% RSLogix 500 project I2P JOB 12-CAYLEN  JOHNSON.RSS, saved by version 10.00.00.00 %
PROJECT "ML06B"    % processor: Bul.1763 MicroLogix 1100 Series B %

PROGRAM FILES
  LAD 2   8 rungs

DATA FILES
  O0 OUTPUT  4 elements
  I1 INPUT  6 elements
  S2 STATUS  66 elements
  B3 BINARY  1 elements
  T4 TIMER  1 elements
  C5 COUNTER  1 elements
  R6 CONTROL  1 elements
  N7 INTEGER  1 elements
  F8 FLOAT  1 elements

LADDER 2
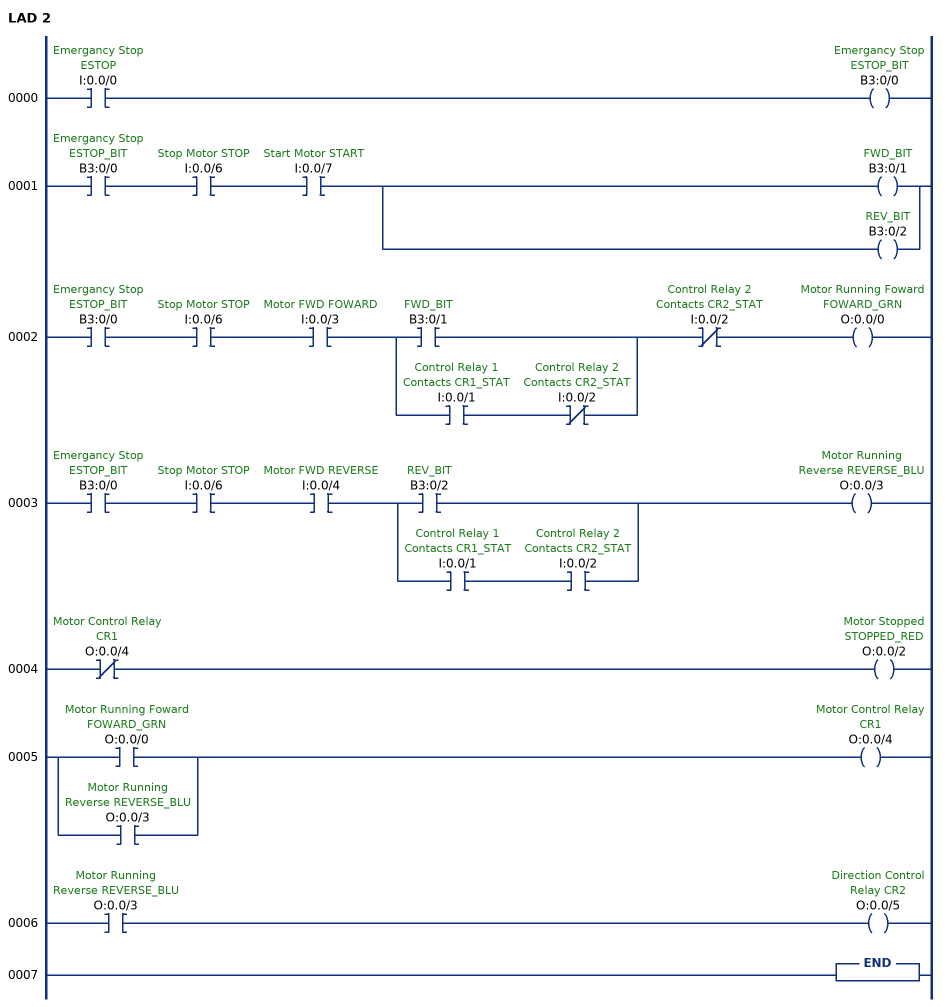
% Rung: 0 %
SOR XIC I:0.0/0 OTE B3:0/0 EOR
%   I:0.0/0  ESTOP  "Emergancy Stop" %
%   B3:0/0  ESTOP_BIT  "Emergancy Stop" %
% Rung: 1 %
SOR XIC B3:0/0 XIC I:0.0/6 XIC I:0.0/7 BST OTE B3:0/1 NXB OTE B3:0/2 BND EOR
%   B3:0/0  ESTOP_BIT  "Emergancy Stop" %
%   I:0.0/6  STOP  "Stop Motor" %
%   I:0.0/7  START  "Start Motor" %
%   B3:0/1  FWD_BIT %
%   B3:0/2  REV_BIT %
% Rung: 2 %
SOR XIC B3:0/0 XIC I:0.0/6 XIC I:0.0/3 BST XIC B3:0/1 NXB XIC I:0.0/1 XIO I:0.0/2 BND XIO I:0.0/2 OTE O:0.0/0 EOR
%   B3:0/0  ESTOP_BIT  "Emergancy Stop" %
%   I:0.0/6  STOP  "Stop Motor" %
%   I:0.0/3  FOWARD  "Motor FWD" %
%   B3:0/1  FWD_BIT %
%   I:0.0/1  CR1_STAT  "Control Relay 1 Contacts" %
%   I:0.0/2  CR2_STAT  "Control Relay 2 Contacts" %
%   O:0.0/0  FOWARD_GRN  "Motor Running Foward" %
% Rung: 3 %
SOR XIC B3:0/0 XIC I:0.0/6 XIC I:0.0/4 BST XIC B3:0/2 NXB XIC I:0.0/1 XIC I:0.0/2 BND OTE O:0.0/3 EOR
%   B3:0/0  ESTOP_BIT  "Emergancy Stop" %
%   I:0.0/6  STOP  "Stop Motor" %
%   I:0.0/4  REVERSE  "Motor FWD" %
%   B3:0/2  REV_BIT %
%   I:0.0/1  CR1_STAT  "Control Relay 1 Contacts" %
%   I:0.0/2  CR2_STAT  "Control Relay 2 Contacts" %
%   O:0.0/3  REVERSE_BLU  "Motor Running Reverse" %
% Rung: 4 %
SOR XIO O:0.0/4 OTE O:0.0/2 EOR
%   O:0.0/4  CR1  "Motor Control Relay" %
%   O:0.0/2  STOPPED_RED  "Motor Stopped" %
% Rung: 5 %
SOR BST XIC O:0.0/0 NXB XIC O:0.0/3 BND OTE O:0.0/4 EOR
%   O:0.0/0  FOWARD_GRN  "Motor Running Foward" %
%   O:0.0/3  REVERSE_BLU  "Motor Running Reverse" %
%   O:0.0/4  CR1  "Motor Control Relay" %
% Rung: 6 %
SOR XIC O:0.0/3 OTE O:0.0/5 EOR
%   O:0.0/3  REVERSE_BLU  "Motor Running Reverse" %
%   O:0.0/5  CR2  "Direction Control Relay" %
% Rung: 7 %
SOR END EOR

OTHER DOCUMENTED ADDRESSES
  I:0.0/5  2PSS_A
  I:0.0/8  PB3  "Push Botton 3"
  O:0.0/1  YLW_LT  "Yellow Light"
  PB1  
